// Mitsubishi GX Works2 project: BookEX6_2 Bitwise   PLC: Q13UDV

// global labels: Global
VAR_GLOBAL
  abArray0 AT M5010 : ARRAY [0..49] OF BOOL;
  sStr0 AT D5000 : STRING[199];
  sStr1 AT D5100 : STRING[199];
  sStr2 AT D5200 : STRING[199];
  sStr3 AT D5300 : STRING[199];
  sStr4 AT D5400 : STRING[199];
  sStr5 AT D5500 : STRING[199];
  sStr6 AT D5600 : STRING[199];
  sStr7 AT D5700 : STRING[199];
  sStr8 AT D5800 : STRING[199];
  sStr9 AT D5900 : STRING[199];
  iVar0 AT D4500 : INT;
  iVar1 AT D4501 : INT;
  iVar2 AT D4502 : INT;
  iVar3 AT D4503 : INT;
  iVar4 AT D4504 : INT;
  iVar5 AT D4505 : INT;
  iVar6 AT D4506 : INT;
  iVar7 AT D4507 : INT;
  iVar8 AT D4508 : INT;
  iVar9 AT D4509 : INT;
  dVar0 AT D4510 : DINT;
  dVar1 AT D4512 : DINT;
  dVar2 AT D4514 : DINT;
  dVar3 AT D4516 : DINT;
  dVar4 AT D4518 : DINT;
  dVar5 AT D4520 : DINT;
  dVar6 AT D4522 : DINT;
  dVar7 AT D4524 : DINT;
  dVar8 AT D4526 : DINT;
  dVar9 AT D4528 : DINT;
  wVar0 AT D4530 : WORD;
  wVar1 AT D4531 : WORD;
  wVar2 AT D4532 : WORD;
  wVar3 AT D4533 : WORD;
  wVar4 AT D4534 : WORD;
  wVar5 AT D4535 : WORD;
  wVar6 AT D4536 : WORD;
  wVar7 AT D4537 : WORD;
  wVar8 AT D4538 : WORD;
  wVar9 AT D4539 : WORD;
  dwVar0 AT D4540 : DWORD;
  dwVar1 AT D4542 : DWORD;
  dwVar2 AT D4544 : DWORD;
  dwVar3 AT D4546 : DWORD;
  dwVar4 AT D4548 : DWORD;
  dwVar5 AT D4550 : DWORD;
  dwVar6 AT D4552 : DWORD;
  dwVar7 AT D4554 : DWORD;
  dwVar8 AT D4556 : DWORD;
  dwVar9 AT D4558 : DWORD;
  fsVar0 AT D4560 : REAL;
  fsVar1 AT D4562 : REAL;
  fsVar2 AT D4564 : REAL;
  fsVar3 AT D4566 : REAL;
  fsVar4 AT D4568 : REAL;
  fsVar5 AT D4570 : REAL;
  fsVar6 AT D4572 : REAL;
  fsVar7 AT D4574 : REAL;
  fsVar8 AT D4576 : REAL;
  fsVar9 AT D4578 : REAL;
  fdVar0 AT D4580 : LREAL;
  tTime0 AT D4620 : TIME;
  tTime1 AT D4622 : TIME;
  tTime2 AT D4624 : TIME;
  tTime3 AT D4626 : TIME;
  tTime4 AT D4628 : TIME;
  tTime5 AT D4630 : TIME;
  tTime6 AT D4632 : TIME;
  tTime7 AT D4634 : TIME;
  tTime8 AT D4636 : TIME;
  tTime9 AT D4638 : TIME;
  tTime10 AT D4640 : TIME;
  bVar0 AT M5000 : BOOL;
  bVar2 AT M5002 : BOOL;
  bVar3 AT M5003 : BOOL;
  bVar4 AT M5004 : BOOL;
  bVar5 AT M5005 : BOOL;
  bVar6 AT M5006 : BOOL;
  bVar7 AT M5007 : BOOL;
  bVar8 AT M5008 : BOOL;
  bVar9 AT M5009 : BOOL;
  abArray1 AT M5060 : ARRAY [0..49] OF BOOL;
  abArray2 AT M5110 : ARRAY [0..49] OF BOOL;
  abArray3 AT M5160 : ARRAY [0..49] OF BOOL;
  abArray4 AT M5210 : ARRAY [0..49] OF BOOL;
  abArray5 AT M5260 : ARRAY [0..49] OF BOOL;
  abArray6 AT M5310 : ARRAY [0..49] OF BOOL;
  abArray7 AT M5360 : ARRAY [0..49] OF BOOL;
  abArray8 AT M5410 : ARRAY [0..49] OF BOOL;
  abArray9 AT M5460 : ARRAY [0..49] OF BOOL;
  fdVar1 AT D4584 : LREAL;
  fdVar2 AT D4588 : LREAL;
  fdVar3 AT D4592 : LREAL;
  fdVar4 AT D4596 : LREAL;
  fdVar5 AT D4600 : LREAL;
  fdVar6 AT D4604 : LREAL;
  fdVar7 AT D4608 : LREAL;
  fdVar8 AT D4612 : LREAL;
  fdVar9 AT D4616 : LREAL;
  adwD10 AT D10 : ARRAY [0..9] OF DWORD;
  awD10 AT D10 : ARRAY [0..19] OF WORD;
  abM10 AT M10 : ARRAY [0..19] OF BOOL;
  bVar1 AT M5001 : BOOL;
END_VAR
// user libraries (not included): HMI

PROGRAM ExBoolFunc
(* structured ladder/FBD written out as ST: instructions are called as NAME(EN, inputs, outputs); _pN, _eN, _tN stand for wires *)
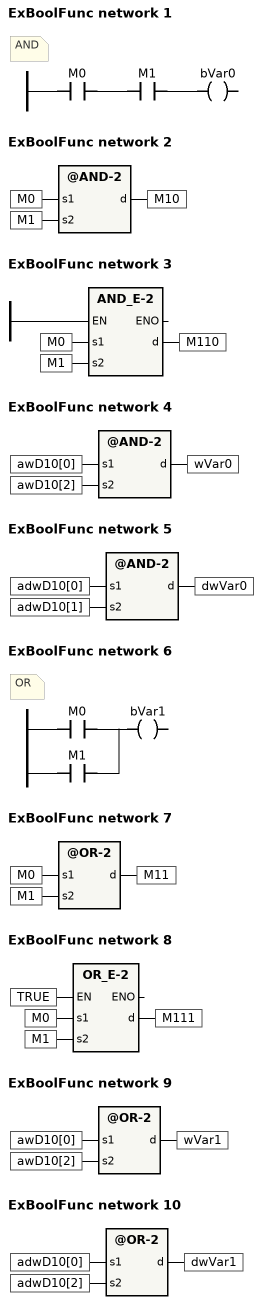
(* network 1 *)
(* AND *)
bVar0 := M0 AND M1;
(* network 2 *)
M10 := @AND-2(M0, M1);
(* network 3 *)
AND_E(TRUE, M0, M1, M110);
(* network 4 *)
wVar0 := @AND-2(awD10[0], awD10[2]);
(* network 5 *)
dwVar0 := @AND-2(adwD10[0], adwD10[1]);
(* network 6 *)
(* OR *)
bVar1 := M0 OR M1;
(* network 7 *)
M11 := @OR-2(M0, M1);
(* network 8 *)
OR_E(TRUE, M0, M1, M111);
(* network 9 *)
wVar1 := @OR-2(awD10[0], awD10[2]);
(* network 10 *)
dwVar1 := @OR-2(adwD10[0], adwD10[2]);
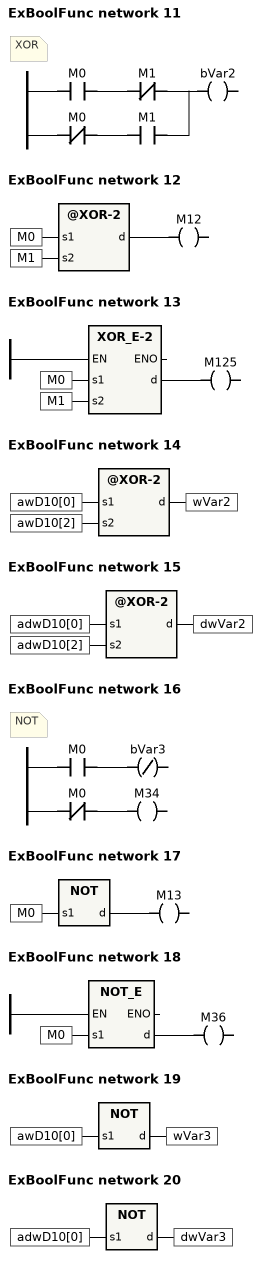
(* network 11 *)
(* XOR *)
bVar2 := (M0 AND NOT M1) OR (NOT M0 AND M1);
(* network 12 *)
M12 := @XOR-2(M0, M1);
(* network 13 *)
XOR_E(TRUE, M0, M1, _t1);
M125 := _t1;
(* network 14 *)
wVar2 := @XOR-2(awD10[0], awD10[2]);
(* network 15 *)
dwVar2 := @XOR-2(adwD10[0], adwD10[2]);
(* network 16 *)
(* NOT *)
bVar3 := NOT M0;
M34 := NOT M0;
(* network 17 *)
M13 := NOT(M0);
(* network 18 *)
NOT_E(TRUE, M0, _t1);
M36 := _t1;
(* network 19 *)
wVar3 := NOT(awD10[0]);
(* network 20 *)
dwVar3 := NOT(adwD10[0]);
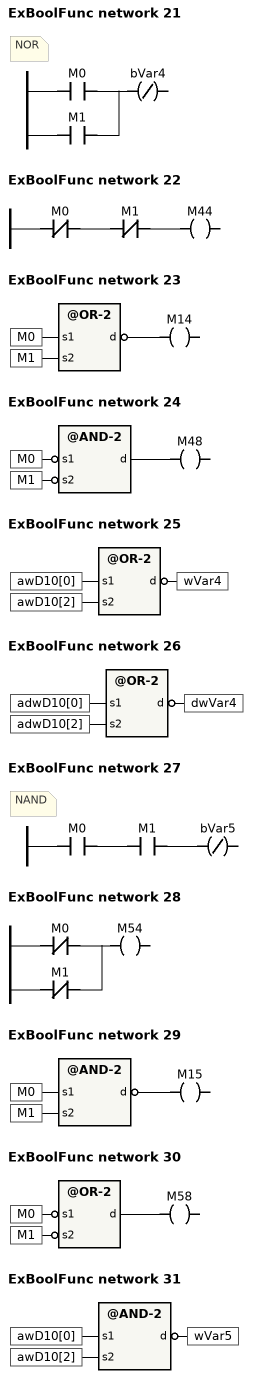
(* network 21 *)
(* NOR *)
bVar4 := NOT (M0 OR M1);
(* network 22 *)
M44 := NOT M0 AND NOT M1;
(* network 23 *)
M14 := NOT (@OR-2(M0, M1));
(* network 24 *)
M48 := @AND-2(NOT M0, NOT M1);
(* network 25 *)
wVar4 := NOT (@OR-2(awD10[0], awD10[2]));
(* network 26 *)
dwVar4 := NOT (@OR-2(adwD10[0], adwD10[2]));
(* network 27 *)
(* NAND *)
bVar5 := NOT (M0 AND M1);
(* network 28 *)
M54 := (NOT M0) OR (NOT M1);
(* network 29 *)
M15 := NOT (@AND-2(M0, M1));
(* network 30 *)
M58 := @OR-2(NOT M0, NOT M1);
(* network 31 *)
wVar5 := NOT (@AND-2(awD10[0], awD10[2]));
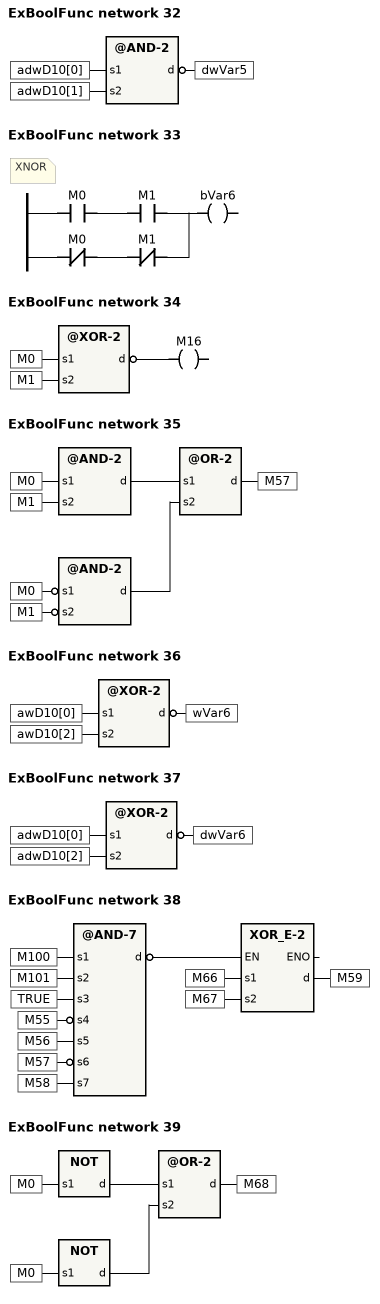
(* network 32 *)
dwVar5 := NOT (@AND-2(adwD10[0], adwD10[1]));
(* network 33 *)
(* XNOR *)
bVar6 := (M0 AND M1) OR (NOT M0 AND NOT M1);
(* network 34 *)
M16 := NOT (@XOR-2(M0, M1));
(* network 35 *)
M57 := @OR-2(@AND-2(M0, M1), @AND-2(NOT M0, NOT M1));
(* network 36 *)
wVar6 := NOT (@XOR-2(awD10[0], awD10[2]));
(* network 37 *)
dwVar6 := NOT (@XOR-2(adwD10[0], adwD10[2]));
(* network 38 *)
XOR_E(NOT (@AND-7(M100, M101, TRUE, NOT M55, M56, NOT M57, M58)), M66, M67, M59);
(* network 39 *)
M68 := @OR-2(NOT(M0), NOT(M0));
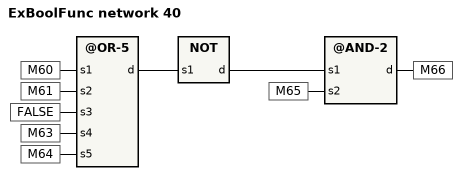
(* network 40 *)
M66 := @AND-2(NOT(@OR-5(M60, M61, FALSE, M63, M64)), M65);
END_PROGRAM

PROGRAM ExBoolFuncST
VAR
  wTemp : ARRAY [0..9] OF WORD;
  dwTemp : ARRAY [0..9] OF DWORD;
END_VAR
;
(* AND *)
M20 := M0 AND M1;
AND_E(TRUE, M0, M1, M220);
wTemp[0] := awD10[0] AND awD10[2];
dwTemp[0] := adwD10[0] AND adwD10[1];

(* OR *)
M21 := M0 OR M1;
OR_E(TRUE, M0, M1, M221);
wTemp[1] := awD10[0] OR awD10[2];
dwTemp[1] := adwD10[0] OR adwD10[1];

(* XOR *)
M22 := M0 XOR M1;
XOR_E(TRUE, M0, M1, M222);
wTemp[2] := awD10[0] XOR awD10[2];
dwTemp[2] := adwD10[0] XOR adwD10[1];

(* NOT *)
M23 := NOT M0;
NOT_E(TRUE, M0, M213);
wTemp[3] := NOT awD10[0];
dwTemp[3] := NOT adwD10[0];

(* NOR *)
M24 := NOT (M0 OR M1);
wTemp[4] := NOT (awD10[0] OR awD10[2]);
dwTemp[4] := NOT (adwD10[0] AND adwD10[1]);

(* NAND *)
M25 := NOT (M0 AND M1);
wTemp[5] := NOT (awD10[0] AND awD10[2]);
dwTemp[5] := NOT (adwD10[0] AND adwD10[1]);

(* XNOR *)
M26 := NOT (M0 XOR M1);
wTemp[6] := NOT (awD10[0] XOR awD10[2]);
dwTemp[6] := NOT (adwD10[0] XOR adwD10[1]);
END_PROGRAM

PROGRAM ExBoolLogic
VAR
  BoolLogic_1 : BoolLogic;
  HMI05_1 : HMI05;
END_VAR
(* structured ladder/FBD written out as ST: instructions are called as NAME(EN, inputs, outputs); _pN, _eN, _tN stand for wires *)
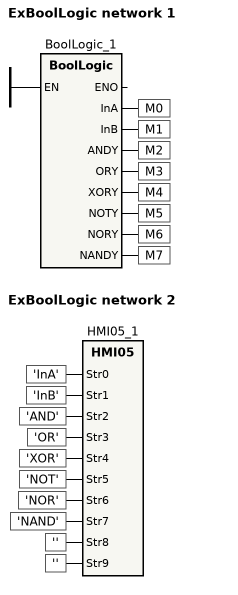
(* network 1 *)
BoolLogic_1(EN := TRUE, InA => M0, InB => M1, ANDY => M2, ORY => M3, XORY => M4, NOTY => M5, NORY => M6, NANDY => M7);
(* network 2 *)
HMI05_1(Str0 := 'InA', Str1 := 'InB', Str2 := 'AND', Str3 := 'OR', Str4 := 'XOR', Str5 := 'NOT', Str6 := 'NOR', Str7 := 'NAND', Str8 := '', Str9 := '');
END_PROGRAM

PROGRAM ExScanInput
VAR
  ScanInput_1 : ScanInput;
  HMI05_1 : HMI05;
END_VAR
(* structured ladder/FBD written out as ST: instructions are called as NAME(EN, inputs, outputs); _pN, _eN, _tN stand for wires *)
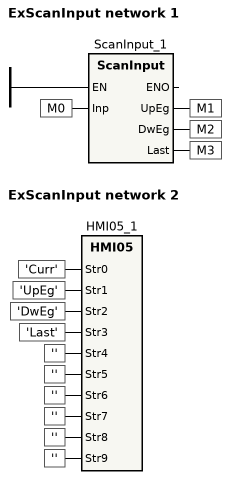
(* network 1 *)
ScanInput_1(EN := TRUE, Inp := M0, UpEg => M1, DwEg => M2, Last => M3);
(* network 2 *)
HMI05_1(Str0 := 'Curr', Str1 := 'UpEg', Str2 := 'DwEg', Str3 := 'Last', Str4 := '', Str5 := '', Str6 := '', Str7 := '', Str8 := '', Str9 := '');
END_PROGRAM

FUNCTION_BLOCK BoolLogic
VAR_OUTPUT
  InA : BOOL;
  InB : BOOL;
END_VAR
VAR
  ScanCnt : INT;
  TmpA : BOOL;
  TmpB : BOOL;
END_VAR
VAR_OUTPUT
  ANDY : BOOL;
  ORY : BOOL;
  XORY : BOOL;
  NOTY : BOOL;
  NORY : BOOL;
  NANDY : BOOL;
END_VAR
;
CASE ScanCnt MOD 4 OF
	0 : TmpA := FALSE;	
	     TmpB := FALSE;
	1 : TmpA := TRUE;	
	     TmpB := FALSE;
	2 : TmpA := FALSE;	
	     TmpB := TRUE;
	3 : TmpA := TRUE;	
	     TmpB := TRUE;
END_CASE;
 
InA := TmpA;
InB := TmpB;
ANDY := InA AND InB;         
ORY := InA OR InB;			 
XORY := InA XOR InB;		 
NOTY := NOT InA;			 
NORY := NOT ORY;
NANDY := NOT ANDY;

ScanCnt := ScanCnt + 1;
END_FUNCTION_BLOCK

FUNCTION Mask
VAR
  Temp : DWORD;
END_VAR
VAR_INPUT
  i_N : INT;
END_VAR
;
CASE i_N OF
	0 : Temp := 0;
	1 : Temp := H00000001;
	2 : Temp := H00000003;
	3 : Temp := H00000007;
	4 : Temp := H0000000F;
	5 : Temp := H0000001F;
	6 : Temp := H0000003F;
	7 : Temp := H0000007F;
	8 : Temp := H000000FF;
	9 : Temp := H000001FF;
	10 : Temp := H000003FF;
	11 : Temp := H000007FF;
	12 : Temp := H00000FFF;
	13 : Temp := H00001FFF;
	14 : Temp := H00003FFF;
	15 : Temp := H00007FFF;
	16 : Temp := H0000FFFF;
	17 : Temp := H0001FFFF;
	18 : Temp := H0003FFFF;
	19 : Temp := H0007FFFF;
	20 : Temp := H000FFFFF;
	21 : Temp := H001FFFFF;
	22 : Temp := H003FFFFF;
	23 : Temp := H007FFFFF;
	24 : Temp := H00FFFFFF;
	25 : Temp := H01FFFFFF;
	26 : Temp := H03FFFFFF;
	27 : Temp := H07FFFFFF;
	28 : Temp := H0FFFFFFF;
	29 : Temp := H1FFFFFFF;
	30 : Temp := H3FFFFFFF;
	31 : Temp := H7FFFFFFF;
	32 : Temp := HFFFFFFFF;
END_CASE;
Mask := Temp;
END_FUNCTION

FUNCTION_BLOCK ScanInput
VAR_INPUT
  Inp : BOOL;
END_VAR
VAR_OUTPUT
  UpEg : BOOL;
END_VAR
VAR
  CurrBit : BOOL;
  LastBit : BOOL;
END_VAR
VAR_OUTPUT
  DwEg : BOOL;
  Last : BOOL;
END_VAR
;
CurrBit := Inp;
UpEg := CurrBit AND NOT LastBit;
DwEg := NOT CurrBit AND LastBit;
Last := LastBit;
LastBit := CurrBit;
END_FUNCTION_BLOCK

FUNCTION_BLOCK W2B_8
VAR_INPUT
  IN : WORD;
END_VAR
VAR_OUTPUT
  Bit0 : BOOL;
  Bit1 : BOOL;
  Bit2 : BOOL;
  Bit3 : BOOL;
  Bit4 : BOOL;
  Bit5 : BOOL;
  Bit6 : BOOL;
  Bit7 : BOOL;
END_VAR
 
Bit0 := (IN AND 16#0001) <> 0;
Bit1 := (IN AND 16#0002) <> 0;
Bit2 := (IN AND 16#0004) <> 0;
Bit3 := (IN AND 16#0008) <> 0;
Bit4 := (IN AND 16#0010) <> 0;
Bit5 := (IN AND 16#0020) <> 0;
Bit6 := (IN AND 16#0040) <> 0;
Bit7 := (IN AND 16#0080) <> 0;
END_FUNCTION_BLOCK

PROGRAM ExW2B8
VAR
  W2B_8_1 : W2B_8;
  W2B_16_1 : W2B_16;
END_VAR
(* structured ladder/FBD written out as ST: instructions are called as NAME(EN, inputs, outputs); _pN, _eN, _tN stand for wires *)
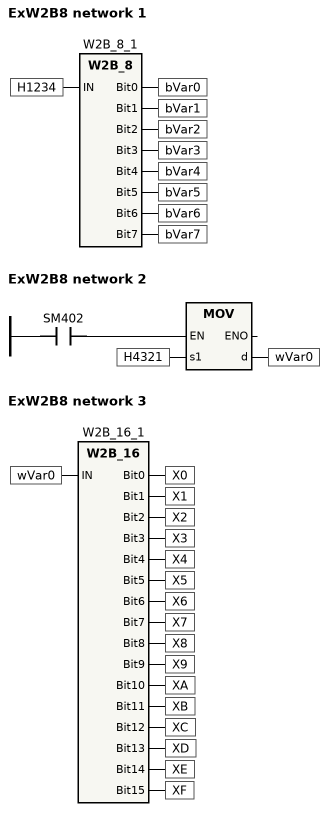
(* network 1 *)
W2B_8_1(IN := H1234, Bit0 => bVar0, Bit1 => bVar1, Bit2 => bVar2, Bit3 => bVar3, Bit4 => bVar4, Bit5 => bVar5, Bit6 => bVar6, Bit7 => bVar7);
(* network 2 *)
MOV(SM402, H4321, wVar0);
(* network 3 *)
W2B_16_1(IN := wVar0, Bit0 => X0, Bit1 => X1, Bit2 => X2, Bit3 => X3, Bit4 => X4, Bit5 => X5, Bit6 => X6, Bit7 => X7, Bit8 => X8, Bit9 => X9, Bit10 => XA, Bit11 => XB, Bit12 => XC, Bit13 => XD, Bit14 => XE, Bit15 => XF);
END_PROGRAM

FUNCTION_BLOCK W2B_16
VAR_INPUT
  IN : WORD;
END_VAR
VAR_OUTPUT
  Bit0 : BOOL;
  Bit1 : BOOL;
  Bit2 : BOOL;
  Bit3 : BOOL;
  Bit4 : BOOL;
  Bit5 : BOOL;
  Bit6 : BOOL;
  Bit7 : BOOL;
  Bit8 : BOOL;
  Bit9 : BOOL;
  Bit10 : BOOL;
  Bit11 : BOOL;
  Bit12 : BOOL;
  Bit13 : BOOL;
  Bit14 : BOOL;
  Bit15 : BOOL;
END_VAR
 
Bit0 := (IN AND 16#0001) <> 0;
Bit1 := (IN AND 16#0002) <> 0;
Bit2 := (IN AND 16#0004) <> 0;
Bit3 := (IN AND 16#0008) <> 0;
Bit4 := (IN AND 16#0010) <> 0;
Bit5 := (IN AND 16#0020) <> 0;
Bit6 := (IN AND 16#0040) <> 0;
Bit7 := (IN AND 16#0080) <> 0;
Bit8 := (IN AND 16#0100) <> 0;
Bit9 := (IN AND 16#0200) <> 0;
Bit10 := (IN AND 16#0400) <> 0;
Bit11 := (IN AND 16#0800) <> 0;
Bit12 := (IN AND 16#1000) <> 0;
Bit13 := (IN AND 16#2000) <> 0;
Bit14 := (IN AND 16#4000) <> 0;
Bit15 := (IN AND 16#8000) <> 0;
END_FUNCTION_BLOCK
